FUNCTION_BLOCK E_DELAY_V (* Composite Function Block Type *)
  (* Standard: 61499-2 *)
  (* Version 0.0, 8/6/2026, Schneider Electric, template *)
  PACKAGE SE.Nereda;
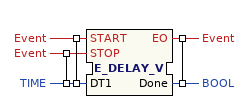
  EVENT_INPUT
    START WITH DT1; (* Begin Delay *)
    STOP WITH DT1; (* Cancel Delay *)
  END_EVENT
  EVENT_OUTPUT
    EO WITH Done;
  END_EVENT
  VAR_INPUT
    DT1 : TIME; (* Delay Time *)
  END_VAR
  VAR_OUTPUT
    Done : BOOL;
  END_VAR
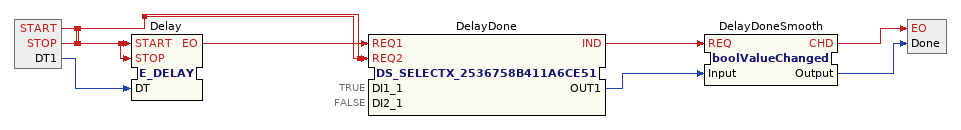
  FBS
    Delay : E_DELAY;
    DelayDone : DS_SELECTX_2536758B411A6CE51(DI1_1 := TRUE, DI2_1 := FALSE); {SET_ATTRIBUTE(Configuration.GenericFBType.InterfaceParams, Runtime.Standard#CNTX:=2;CNTY:=1;DI${CNTX,_,CNTY$}:BOOL)}
    DelayDoneSmooth : boolValueChanged;
  END_FBS
  EVENT_CONNECTIONS
    START TO Delay.START;
    STOP TO Delay.STOP;
    Delay.EO TO DelayDone.REQ1;
    DelayDone.IND TO DelayDoneSmooth.REQ;
    DelayDoneSmooth.CHD TO EO;
    START TO DelayDone.REQ2;
    STOP TO DelayDone.REQ2;
  END_CONNECTIONS
  DATA_CONNECTIONS
    DT1 TO Delay.DT;
    DelayDone.OUT1 TO DelayDoneSmooth.Input;
    DelayDoneSmooth.Output TO Done;
  END_CONNECTIONS
END_FUNCTION_BLOCK
